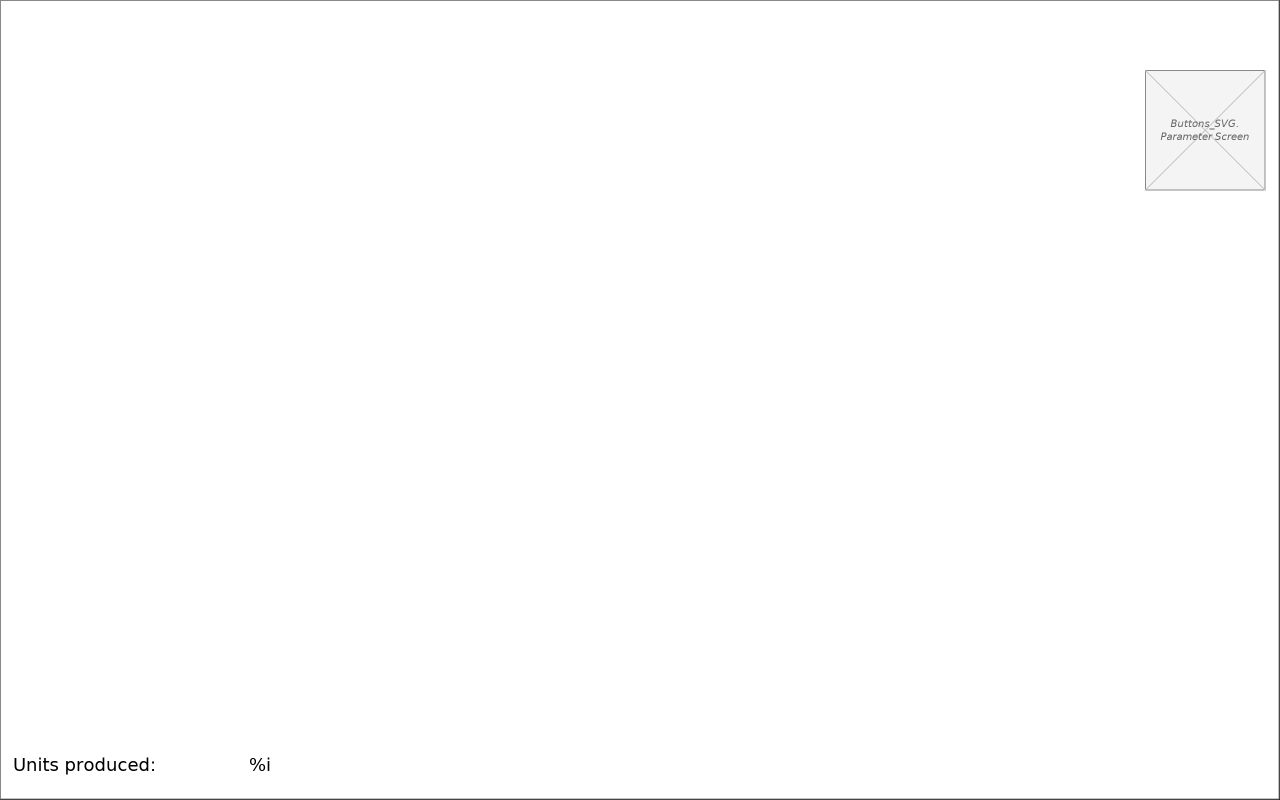
VISUALIZATION Settings  // 1280x800
VAR_IN_OUT
	bCmdParameter : BOOL ; // Go to parameter screen
	nUnitsProduced : UDINT ; // Units produced in machine lifetime
END_VAR
    Rectangle (0,0 1280x800)
    Label (10,750 150x30), "Units produced:"
    Textfield (160,750 200x30), "%i", text variable: nUnitsProduced
    Image (1145,70 120x120), image: Buttons_SVG.Parameter Screen
        OnMouseClick: toggle bCmdParameter
END_VISUALIZATION

(* stored: Version 1.1.0.1, ProductVersion 3.1.4024.5
   Visu Settings: Id {4270b803-3409-4185-bb86-fbae2b2398e9} *)
